// TIA Portal V17 export
// export: Created 2023-04-03T06:31:32.4476947Z, ExportSetting WithDefaults, DisplayName Totally Integrated Automation Portal, DisplayVersion V17 Update 4, DisplayName TIA Portal Openness, DisplayVersion V17 Update 4, DisplayName TIA Portal Version Control Interface, DisplayVersion V17, DisplayName STEP 7 Professional, DisplayVersion V17 Update 4, DisplayName STEP 7 Safety, DisplayVersion V17, DisplayName WinCC Professional, DisplayVersion V17 Update 4
DATA_BLOCK "HMI"   // DB110
{ S7_Optimized_Access := 'TRUE' }
VERSION : 0.1
// stored: AutoNumber false, DBAccessibleFromOPCUA true, DBAccessibleFromWebserver true, IsOnlyStoredInLoadMemory false, IsRetainMemResEnabled false, IsWriteProtectedInAS false, MemoryReserve 100
   VAR
      SS1 : Struct
         xLocalCmd : Bool;
         xEnbCmd : Bool := True;
         xLocalSt : Bool;
         rPacRef : Real;
         rQacRef : Real;
      END_STRUCT;
      SS2 : Struct
         xLocalCmd : Bool;
         xEnbCmd : Bool := True;
         xLocalSt : Bool;
         rPacRef : Real;
         rQacRef : Real;
      END_STRUCT;
      xLocalCmd : Bool;
      xStopCmd : Bool;
      xStandByCmd : Bool;
      xRunCmd : Bool;
      xTestCmd : Bool;
      xLocalSt : Bool;
      xStopSt : Bool;
      xStandBySt : Bool;
      xRunSt : Bool;
      rPacAutomRef : Real;
      PCS1 : Struct
         xEnbDCbus1 : Bool := True;
         xEnbDCbus2 : Bool := True;
      END_STRUCT;
      iNMaxRackFault : Int := 1;
      iNMinRackEnable : Int := 1;
      rSnPE : Real;
      xBB1BR1AlmDisable : Bool;
      xBB1BR2AlmDisable : Bool;
      xBB1BR3AlmDisable : Bool;
      xBB1BR4AlmDisable : Bool;
      xBB1BR5AlmDisable : Bool;
      xBB1BR6AlmDisable : Bool;
      xBB1BR7AlmDisable : Bool;
      xBB1BR8AlmDisable : Bool;
      xBB1BR9AlmDisable : Bool;
      xBB1BR10AlmDisable : Bool;
      xBB2BR1AlmDisable : Bool;
      xBB2BR2AlmDisable : Bool;
      xBB2BR3AlmDisable : Bool;
      xBB2BR4AlmDisable : Bool;
      xBB2BR5AlmDisable : Bool;
      xBB2BR6AlmDisable : Bool;
      xBB2BR7AlmDisable : Bool;
      xBB2BR8AlmDisable : Bool;
      xBB2BR9AlmDisable : Bool;
      xBB2BR10AlmDisable : Bool;
      xBB1AlmDisable : Bool;
      xBB2AlmDisable : Bool;
      xPEMSAlmDisable : Bool;
      xPCSAlmDisable : Bool;
      xMVSkidAlmDisable : Bool;
      xPIAlmDisable : Bool;
   END_VAR
BEGIN
END_DATA_BLOCK
